// TIA Portal V16 export
// export: Created 2021-07-12T14:47:21.3421368Z, ExportSetting WithDefaults, DisplayName Totally Integrated Automation Portal, DisplayVersion V16, DisplayName TIA Portal Version Control Interface, DisplayVersion V16, DisplayName TIA Portal Openness, DisplayVersion V16, DisplayName STEP 7 Professional, DisplayVersion V16, DisplayName STEP 7 Safety, DisplayVersion V16, DisplayName WinCC Professional, DisplayVersion V16
TYPE "SimaHydTO_typeHMIConnectionParameterSettingsAxisData"
TITLE = SimaHydTO_typeHMIConnectionParameterSettingsAxisData
// Axis data
// stored: IsFailsafeCompliant false
   STRUCT
      Actor { S7_SetPoint := 'True'} : "LSimaHydTO_typeActor";   // Actor configuration
      ValveCharacteristic { S7_SetPoint := 'True'} : "LSimaHydTO_typeValveCharacteristic";   // Valve characteristic
      ForceLimits { S7_SetPoint := 'True'} : "LSimaHydTO_typeForceLimits";   // Force limits
      Pressure_A_Transducer { S7_SetPoint := 'True'} : "LSimaHydTO_typeTransducer";   // Piston side pressure transducer configuration
      Pressure_B_Transducer { S7_SetPoint := 'True'} : "LSimaHydTO_typeTransducer";   // Piston rod side pressure transducer configuration
      PositionControl { S7_SetPoint := 'True'} : "LSimaHydTO_typePositionControl";   // Position control configuration data
      ForceControl { S7_SetPoint := 'True'} : "LSimaHydTO_typeForceControl";   // Force control configuration data
      DynamicAxisModel { S7_SetPoint := 'True'} : "LSimaHydTO_typeDynamicAxisModel";   // Settings of the balancing filter
      SmoothingFilter { S7_SetPoint := 'True'} : "LSimaHydTO_typeSmoothingFilter";   // Settings of the smoothing filter
      StatusActor { S7_SetPoint := 'True'} : "LSimaHydTO_typeStatusActor";   // Indicates the status of actor data
      StatusVChar { S7_SetPoint := 'True'} : "LSimaHydTO_typeStatusVChar";   // Indicates the status of valve characteristic data
      Status_A_Transducer { S7_SetPoint := 'True'} : "LSimaHydTO_typeStatusTransducer";   // Indicates the status of piston side pressure transducer data
      Status_B_Transducer { S7_SetPoint := 'True'} : "LSimaHydTO_typeStatusTransducer";   // Indicates the status of piston rod side pressure transducer data
      StatusServo { S7_SetPoint := 'True'} : "LSimaHydTO_typeStatusServo";   // Indicates the status of position control
      StatusForce { S7_SetPoint := 'True'} : "LSimaHydTO_typeStatusForce";   // Indicates the status of force control
      StatusForceProfile { S7_SetPoint := 'True'} : "LSimaHydTO_typeStatusForceProfile";   // Indicates the status of a force profile processing
      "Name" : WString[24];   // Name displayed on HMI
      VCharName : WString[24];   // Charachteristic name displayed on HMI
   END_STRUCT;
END_TYPE
